(* Logix 5000 project; controller SX_V040001_C001 vendor 1 type 14 code 77 rev 16.23; software revision 16.04; part 27 of 35 *)
(* tags used below, declared in another part *)
   ALL_KINDS : INT[90];
   loading : INT[19];
   METERING : INT[44];
   NOTDOS : INT[6];
   PARAMETER : INT[501];
   T_DELTA_EM_METER : TIMER;
(* MainProgram, continued *)

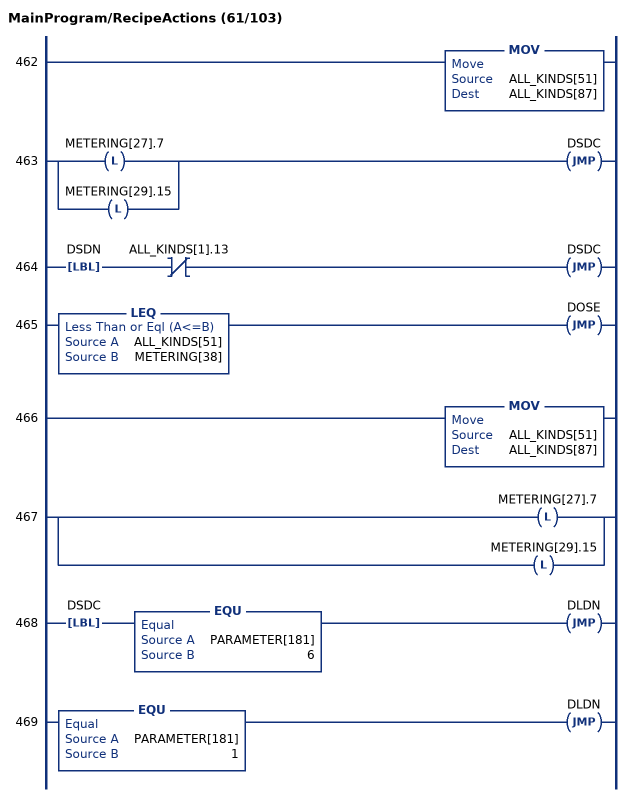
   [picture p595: MainProgram/RecipeActions rungs 462-469]
   462: MOV(ALL_KINDS[51],ALL_KINDS[87]);
   463: [OTL(METERING[27].7) ,OTL(METERING[29].15) ]JMP(DSDC);
   464: LBL(DSDN)XIO(ALL_KINDS[1].13)JMP(DSDC);
   465: LEQ(ALL_KINDS[51],METERING[38])JMP(DOSE);
   466: MOV(ALL_KINDS[51],ALL_KINDS[87]);
   467: [OTL(METERING[27].7) ,OTL(METERING[29].15) ];
   468: LBL(DSDC)EQU(PARAMETER[181],6)JMP(DLDN);
   469: EQU(PARAMETER[181],1)JMP(DLDN);
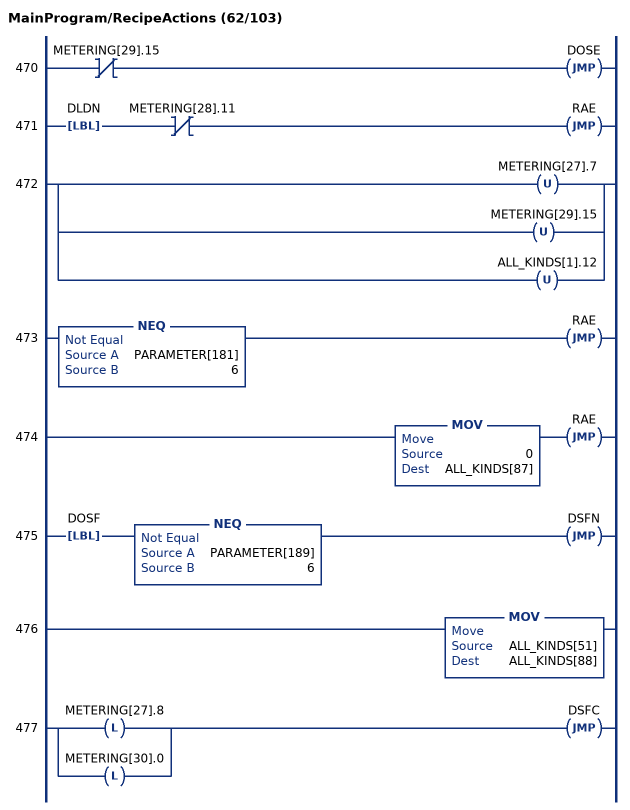
   470: XIO(METERING[29].15)JMP(DOSE);
   471: LBL(DLDN)XIO(METERING[28].11)JMP(RAE);
   472: [OTU(METERING[27].7) ,OTU(METERING[29].15) ,OTU(ALL_KINDS[1].12) ];
   473: NEQ(PARAMETER[181],6)JMP(RAE);
   474: MOV(0,ALL_KINDS[87])JMP(RAE);
   475: LBL(DOSF)NEQ(PARAMETER[189],6)JMP(DSFN);
   476: MOV(ALL_KINDS[51],ALL_KINDS[88]);
   477: [OTL(METERING[27].8) ,OTL(METERING[30].0) ]JMP(DSFC);
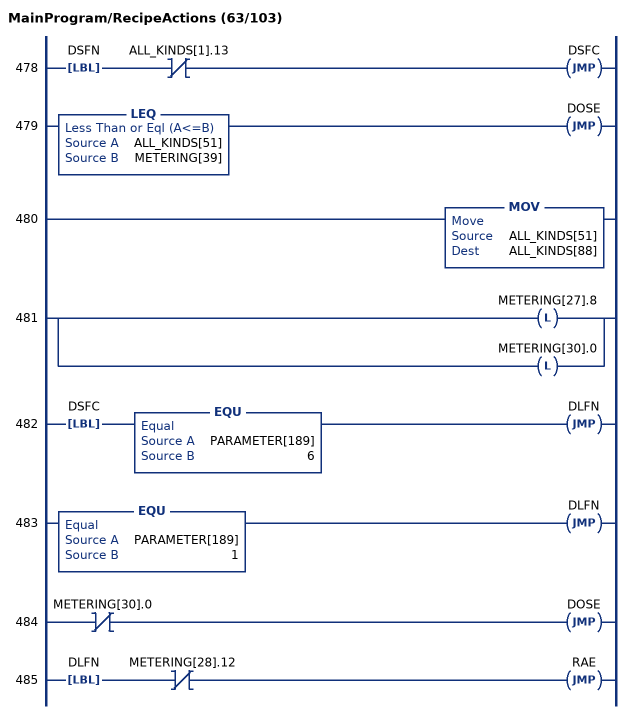
   478: LBL(DSFN)XIO(ALL_KINDS[1].13)JMP(DSFC);
   479: LEQ(ALL_KINDS[51],METERING[39])JMP(DOSE);
   480: MOV(ALL_KINDS[51],ALL_KINDS[88]);
   481: [OTL(METERING[27].8) ,OTL(METERING[30].0) ];
   482: LBL(DSFC)EQU(PARAMETER[189],6)JMP(DLFN);
   483: EQU(PARAMETER[189],1)JMP(DLFN);
   484: XIO(METERING[30].0)JMP(DOSE);
   485: LBL(DLFN)XIO(METERING[28].12)JMP(RAE);
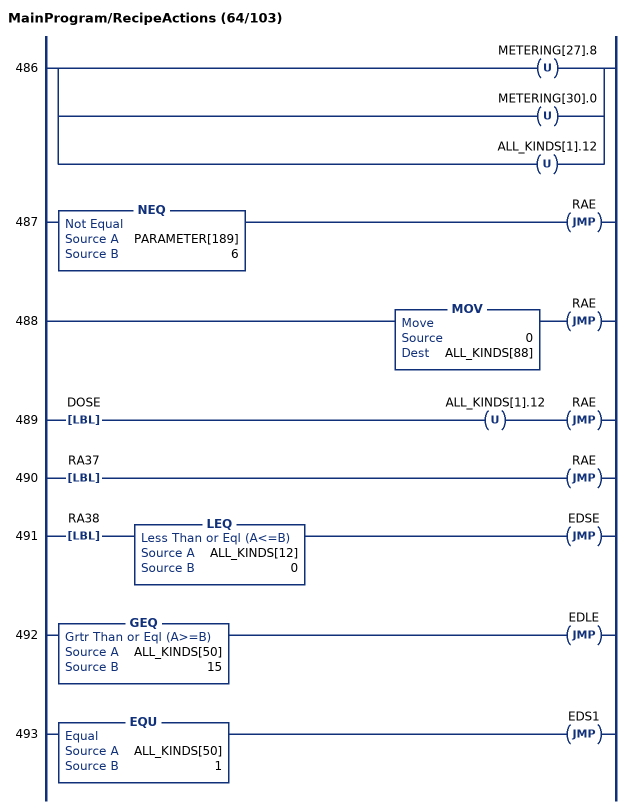
   486: [OTU(METERING[27].8) ,OTU(METERING[30].0) ,OTU(ALL_KINDS[1].12) ];
   487: NEQ(PARAMETER[189],6)JMP(RAE);
   488: MOV(0,ALL_KINDS[88])JMP(RAE);
   489: LBL(DOSE)OTU(ALL_KINDS[1].12)JMP(RAE);
   490: LBL(RA37)JMP(RAE);
   491: LBL(RA38)LEQ(ALL_KINDS[12],0)JMP(EDSE);
   492: GEQ(ALL_KINDS[50],15)JMP(EDLE);
   493: EQU(ALL_KINDS[50],1)JMP(EDS1);
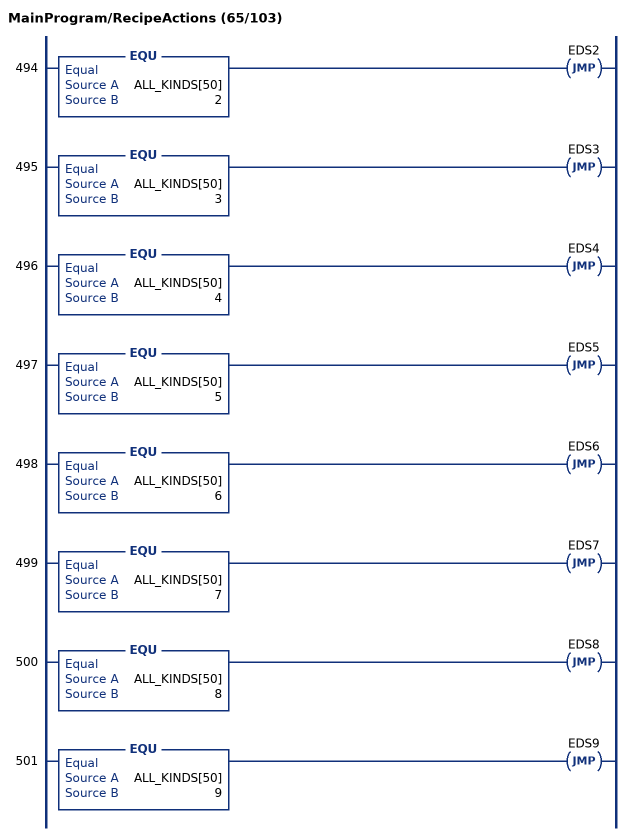
   494: EQU(ALL_KINDS[50],2)JMP(EDS2);
   495: EQU(ALL_KINDS[50],3)JMP(EDS3);
   496: EQU(ALL_KINDS[50],4)JMP(EDS4);
   497: EQU(ALL_KINDS[50],5)JMP(EDS5);
   498: EQU(ALL_KINDS[50],6)JMP(EDS6);
   499: EQU(ALL_KINDS[50],7)JMP(EDS7);
   500: EQU(ALL_KINDS[50],8)JMP(EDS8);
   501: EQU(ALL_KINDS[50],9)JMP(EDS9);
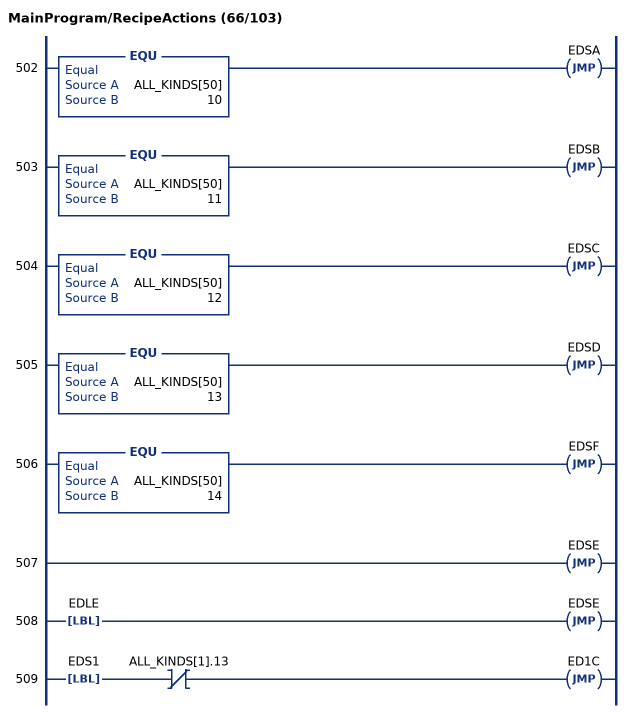
   502: EQU(ALL_KINDS[50],10)JMP(EDSA);
   503: EQU(ALL_KINDS[50],11)JMP(EDSB);
   504: EQU(ALL_KINDS[50],12)JMP(EDSC);
   505: EQU(ALL_KINDS[50],13)JMP(EDSD);
   506: EQU(ALL_KINDS[50],14)JMP(EDSF);
   507: JMP(EDSE);
   508: LBL(EDLE)JMP(EDSE);
   509: LBL(EDS1)XIO(ALL_KINDS[1].13)JMP(ED1C);
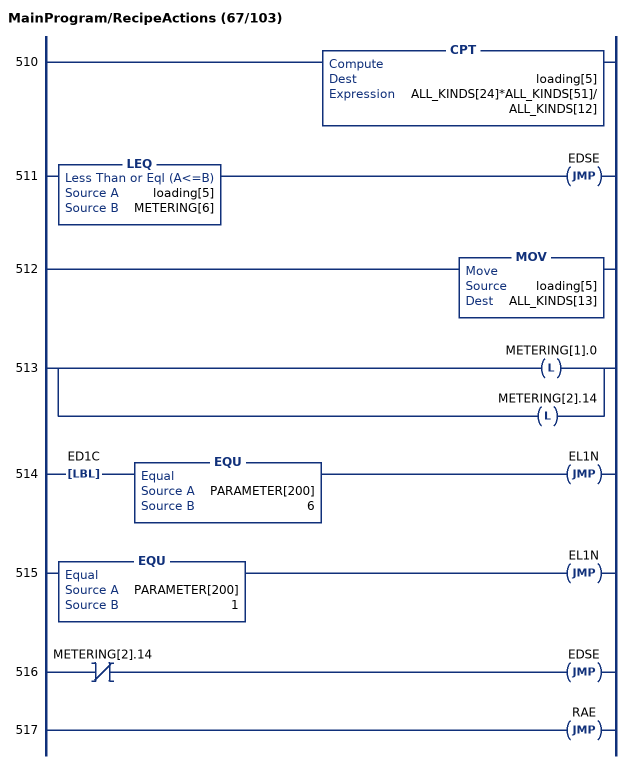
   510: CPT(loading[5],ALL_KINDS[24]*ALL_KINDS[51]/ALL_KINDS[12]);
   511: LEQ(loading[5],METERING[6])JMP(EDSE);
   512: MOV(loading[5],ALL_KINDS[13]);
   513: [OTL(METERING[1].0) ,OTL(METERING[2].14) ];
   514: LBL(ED1C)EQU(PARAMETER[200],6)JMP(EL1N);
   515: EQU(PARAMETER[200],1)JMP(EL1N);
   516: XIO(METERING[2].14)JMP(EDSE);
   517: JMP(RAE);
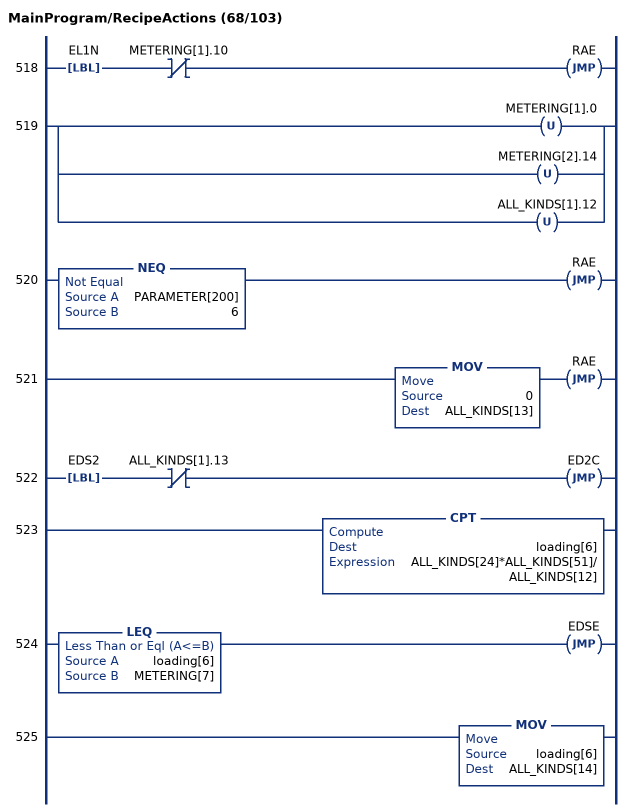
   518: LBL(EL1N)XIO(METERING[1].10)JMP(RAE);
   519: [OTU(METERING[1].0) ,OTU(METERING[2].14) ,OTU(ALL_KINDS[1].12) ];
   520: NEQ(PARAMETER[200],6)JMP(RAE);
   521: MOV(0,ALL_KINDS[13])JMP(RAE);
   522: LBL(EDS2)XIO(ALL_KINDS[1].13)JMP(ED2C);
   523: CPT(loading[6],ALL_KINDS[24]*ALL_KINDS[51]/ALL_KINDS[12]);
   524: LEQ(loading[6],METERING[7])JMP(EDSE);
   525: MOV(loading[6],ALL_KINDS[14]);
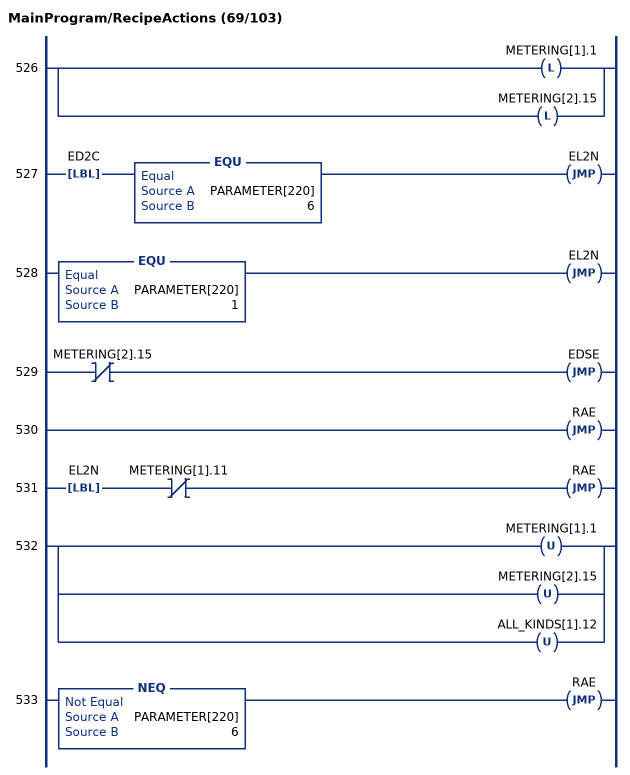
   526: [OTL(METERING[1].1) ,OTL(METERING[2].15) ];
   527: LBL(ED2C)EQU(PARAMETER[220],6)JMP(EL2N);
   528: EQU(PARAMETER[220],1)JMP(EL2N);
   529: XIO(METERING[2].15)JMP(EDSE);
   530: JMP(RAE);
   531: LBL(EL2N)XIO(METERING[1].11)JMP(RAE);
   532: [OTU(METERING[1].1) ,OTU(METERING[2].15) ,OTU(ALL_KINDS[1].12) ];
   533: NEQ(PARAMETER[220],6)JMP(RAE);
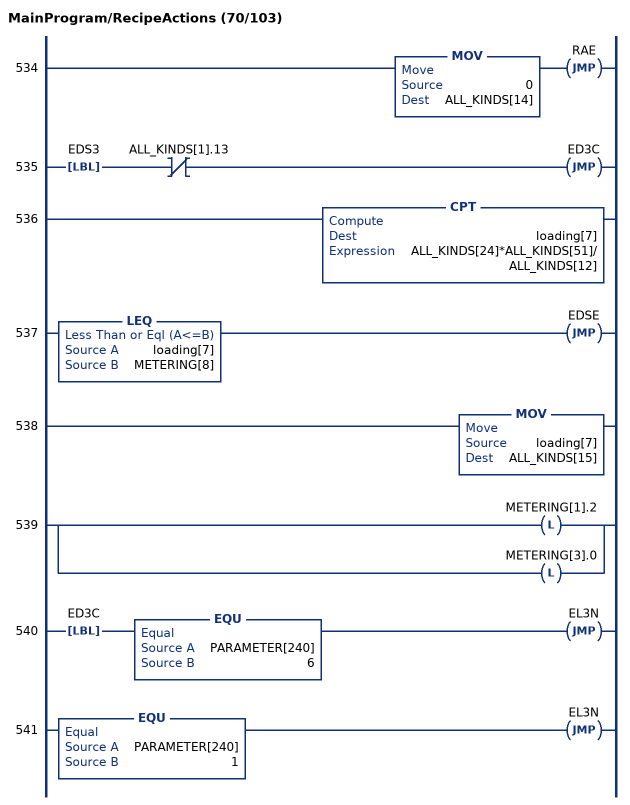
   534: MOV(0,ALL_KINDS[14])JMP(RAE);
   535: LBL(EDS3)XIO(ALL_KINDS[1].13)JMP(ED3C);
   536: CPT(loading[7],ALL_KINDS[24]*ALL_KINDS[51]/ALL_KINDS[12]);
   537: LEQ(loading[7],METERING[8])JMP(EDSE);
   538: MOV(loading[7],ALL_KINDS[15]);
   539: [OTL(METERING[1].2) ,OTL(METERING[3].0) ];
   540: LBL(ED3C)EQU(PARAMETER[240],6)JMP(EL3N);
   541: EQU(PARAMETER[240],1)JMP(EL3N);
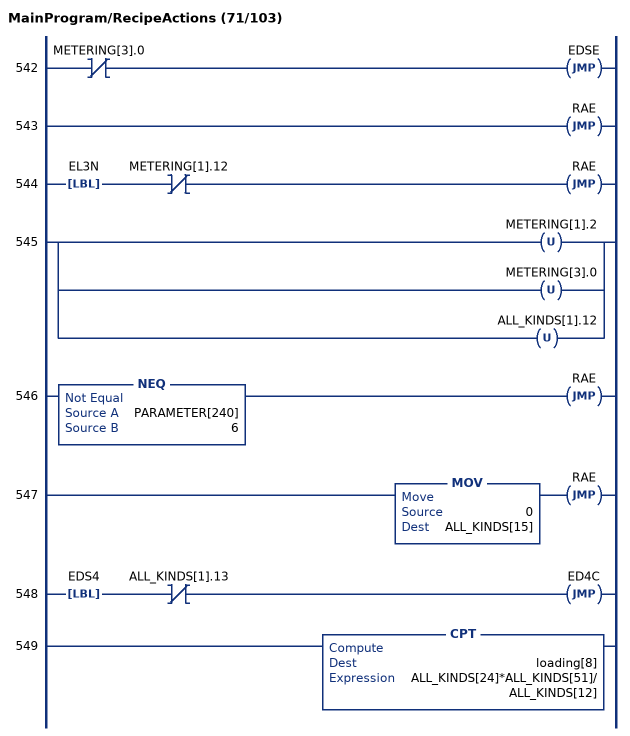
   542: XIO(METERING[3].0)JMP(EDSE);
   543: JMP(RAE);
   544: LBL(EL3N)XIO(METERING[1].12)JMP(RAE);
   545: [OTU(METERING[1].2) ,OTU(METERING[3].0) ,OTU(ALL_KINDS[1].12) ];
   546: NEQ(PARAMETER[240],6)JMP(RAE);
   547: MOV(0,ALL_KINDS[15])JMP(RAE);
   548: LBL(EDS4)XIO(ALL_KINDS[1].13)JMP(ED4C);
   549: CPT(loading[8],ALL_KINDS[24]*ALL_KINDS[51]/ALL_KINDS[12]);
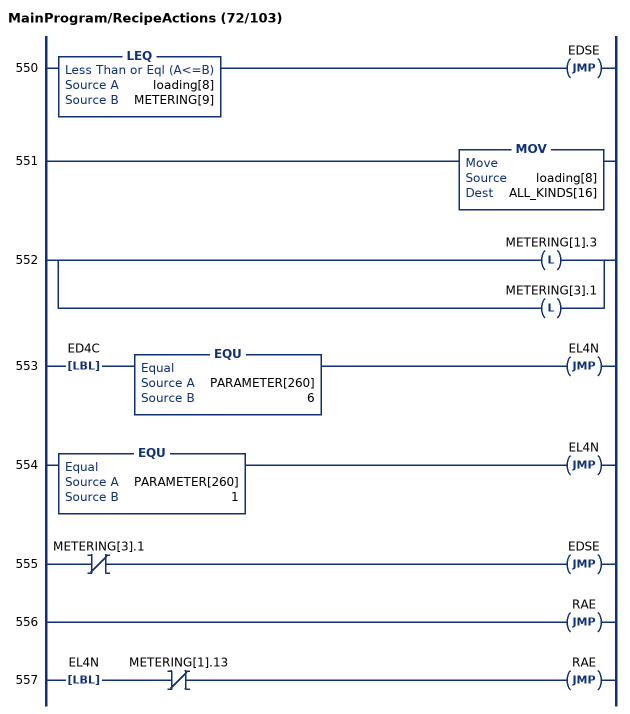
   550: LEQ(loading[8],METERING[9])JMP(EDSE);
   551: MOV(loading[8],ALL_KINDS[16]);
   552: [OTL(METERING[1].3) ,OTL(METERING[3].1) ];
   553: LBL(ED4C)EQU(PARAMETER[260],6)JMP(EL4N);
   554: EQU(PARAMETER[260],1)JMP(EL4N);
   555: XIO(METERING[3].1)JMP(EDSE);
   556: JMP(RAE);
   557: LBL(EL4N)XIO(METERING[1].13)JMP(RAE);
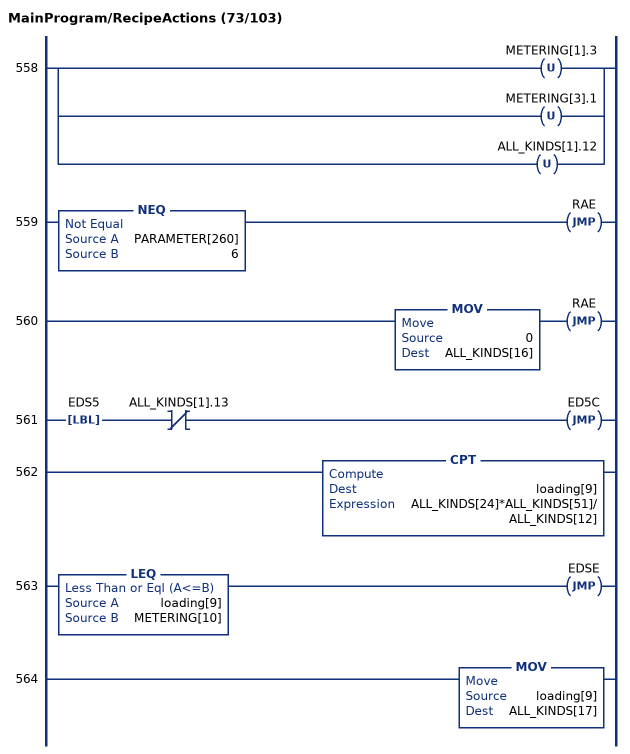
   558: [OTU(METERING[1].3) ,OTU(METERING[3].1) ,OTU(ALL_KINDS[1].12) ];
   559: NEQ(PARAMETER[260],6)JMP(RAE);
   560: MOV(0,ALL_KINDS[16])JMP(RAE);
   561: LBL(EDS5)XIO(ALL_KINDS[1].13)JMP(ED5C);
   562: CPT(loading[9],ALL_KINDS[24]*ALL_KINDS[51]/ALL_KINDS[12]);
   563: LEQ(loading[9],METERING[10])JMP(EDSE);
   564: MOV(loading[9],ALL_KINDS[17]);
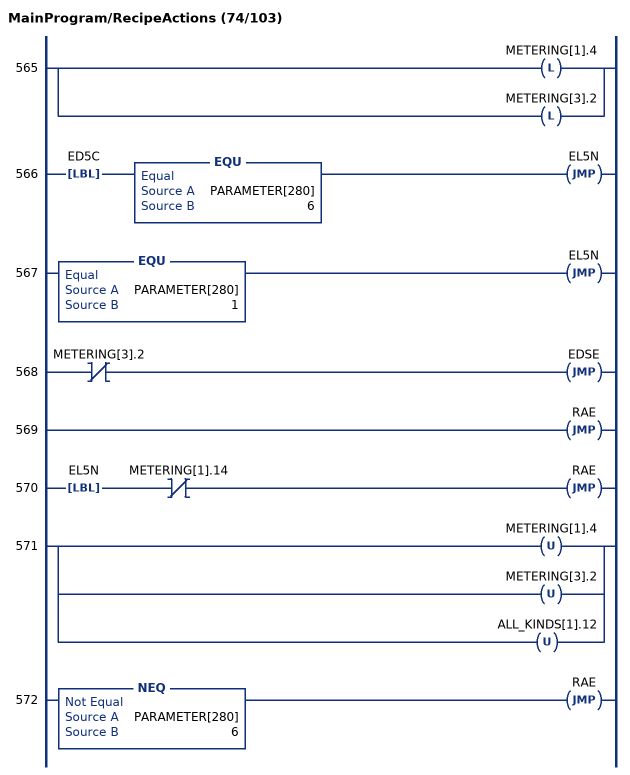
   565: [OTL(METERING[1].4) ,OTL(METERING[3].2) ];
   566: LBL(ED5C)EQU(PARAMETER[280],6)JMP(EL5N);
   567: EQU(PARAMETER[280],1)JMP(EL5N);
   568: XIO(METERING[3].2)JMP(EDSE);
   569: JMP(RAE);
   570: LBL(EL5N)XIO(METERING[1].14)JMP(RAE);
   571: [OTU(METERING[1].4) ,OTU(METERING[3].2) ,OTU(ALL_KINDS[1].12) ];
   572: NEQ(PARAMETER[280],6)JMP(RAE);
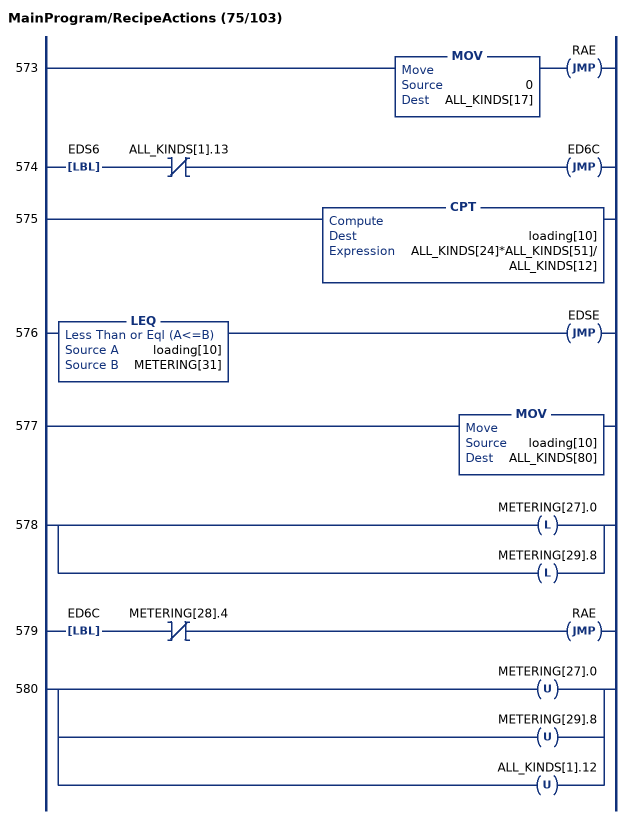
   573: MOV(0,ALL_KINDS[17])JMP(RAE);
   574: LBL(EDS6)XIO(ALL_KINDS[1].13)JMP(ED6C);
   575: CPT(loading[10],ALL_KINDS[24]*ALL_KINDS[51]/ALL_KINDS[12]);
   576: LEQ(loading[10],METERING[31])JMP(EDSE);
   577: MOV(loading[10],ALL_KINDS[80]);
   578: [OTL(METERING[27].0) ,OTL(METERING[29].8) ];
   579: LBL(ED6C)XIO(METERING[28].4)JMP(RAE);
   580: [OTU(METERING[27].0) ,OTU(METERING[29].8) ,OTU(ALL_KINDS[1].12) ];
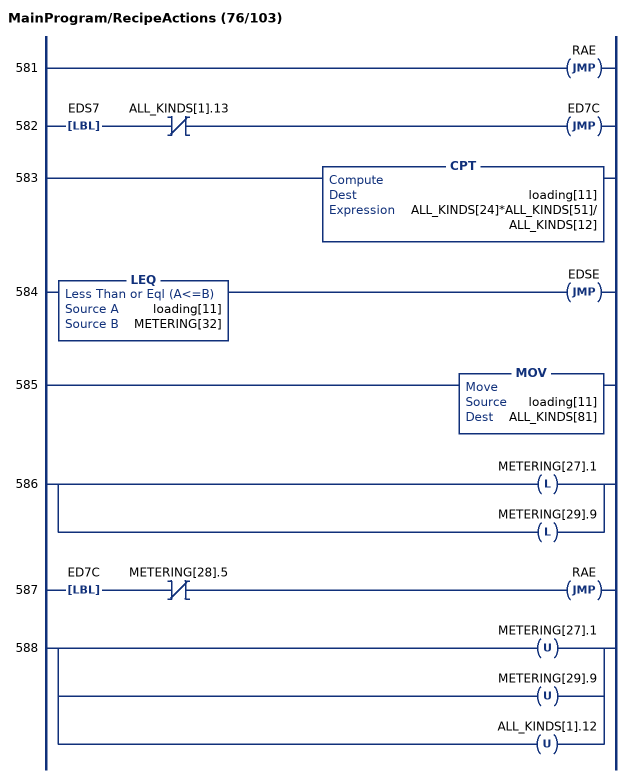
   581: JMP(RAE);
   582: LBL(EDS7)XIO(ALL_KINDS[1].13)JMP(ED7C);
   583: CPT(loading[11],ALL_KINDS[24]*ALL_KINDS[51]/ALL_KINDS[12]);
   584: LEQ(loading[11],METERING[32])JMP(EDSE);
   585: MOV(loading[11],ALL_KINDS[81]);
   586: [OTL(METERING[27].1) ,OTL(METERING[29].9) ];
   587: LBL(ED7C)XIO(METERING[28].5)JMP(RAE);
   588: [OTU(METERING[27].1) ,OTU(METERING[29].9) ,OTU(ALL_KINDS[1].12) ];
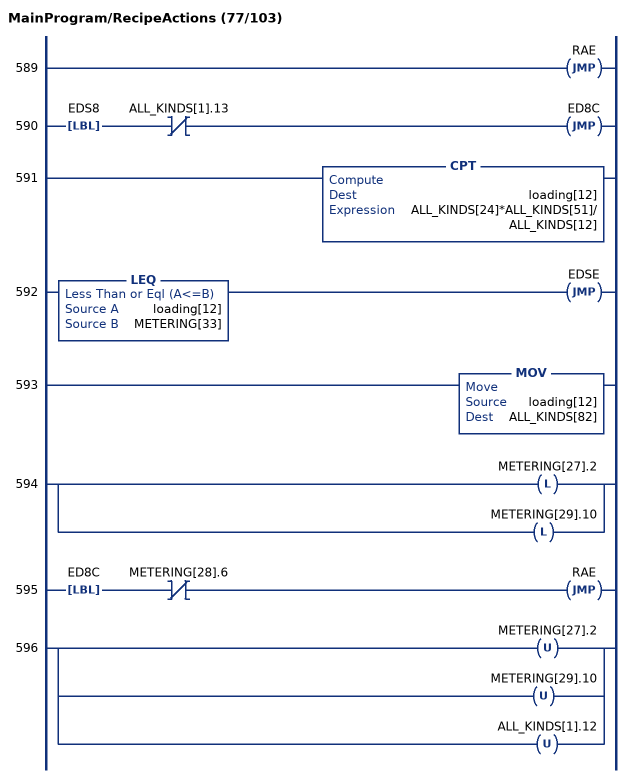
   589: JMP(RAE);
   590: LBL(EDS8)XIO(ALL_KINDS[1].13)JMP(ED8C);
   591: CPT(loading[12],ALL_KINDS[24]*ALL_KINDS[51]/ALL_KINDS[12]);
   592: LEQ(loading[12],METERING[33])JMP(EDSE);
   593: MOV(loading[12],ALL_KINDS[82]);
   594: [OTL(METERING[27].2) ,OTL(METERING[29].10) ];
   595: LBL(ED8C)XIO(METERING[28].6)JMP(RAE);
   596: [OTU(METERING[27].2) ,OTU(METERING[29].10) ,OTU(ALL_KINDS[1].12) ];
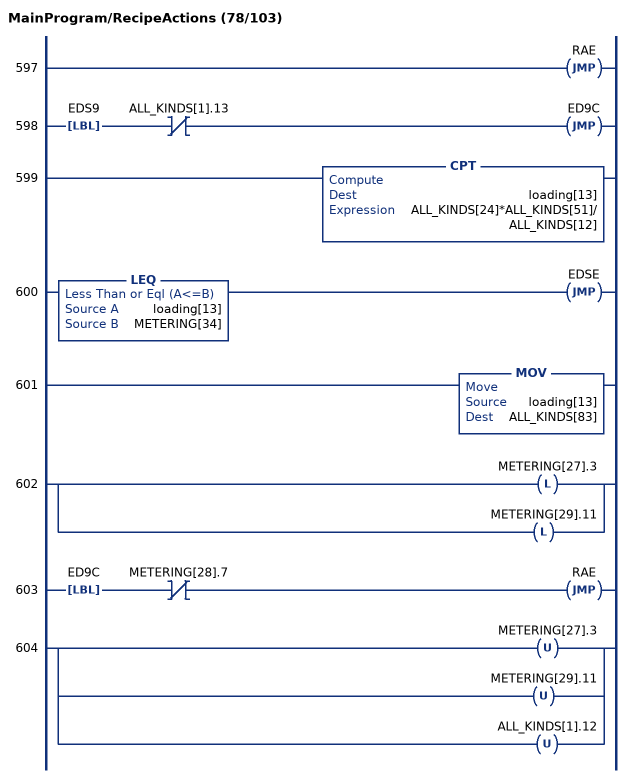
   597: JMP(RAE);
   598: LBL(EDS9)XIO(ALL_KINDS[1].13)JMP(ED9C);
   599: CPT(loading[13],ALL_KINDS[24]*ALL_KINDS[51]/ALL_KINDS[12]);
   600: LEQ(loading[13],METERING[34])JMP(EDSE);
   601: MOV(loading[13],ALL_KINDS[83]);
   602: [OTL(METERING[27].3) ,OTL(METERING[29].11) ];
   603: LBL(ED9C)XIO(METERING[28].7)JMP(RAE);
   604: [OTU(METERING[27].3) ,OTU(METERING[29].11) ,OTU(ALL_KINDS[1].12) ];
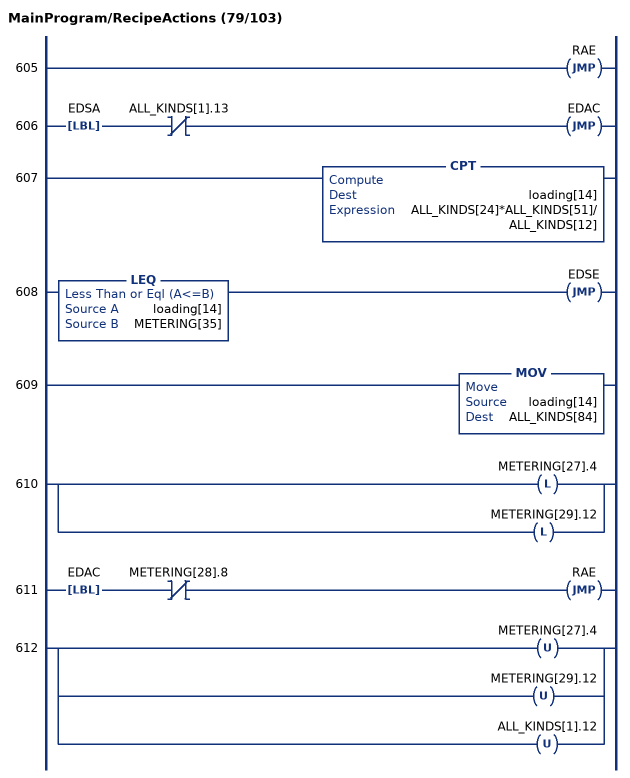
   605: JMP(RAE);
   606: LBL(EDSA)XIO(ALL_KINDS[1].13)JMP(EDAC);
   607: CPT(loading[14],ALL_KINDS[24]*ALL_KINDS[51]/ALL_KINDS[12]);
   608: LEQ(loading[14],METERING[35])JMP(EDSE);
   609: MOV(loading[14],ALL_KINDS[84]);
   610: [OTL(METERING[27].4) ,OTL(METERING[29].12) ];
   611: LBL(EDAC)XIO(METERING[28].8)JMP(RAE);
   612: [OTU(METERING[27].4) ,OTU(METERING[29].12) ,OTU(ALL_KINDS[1].12) ];
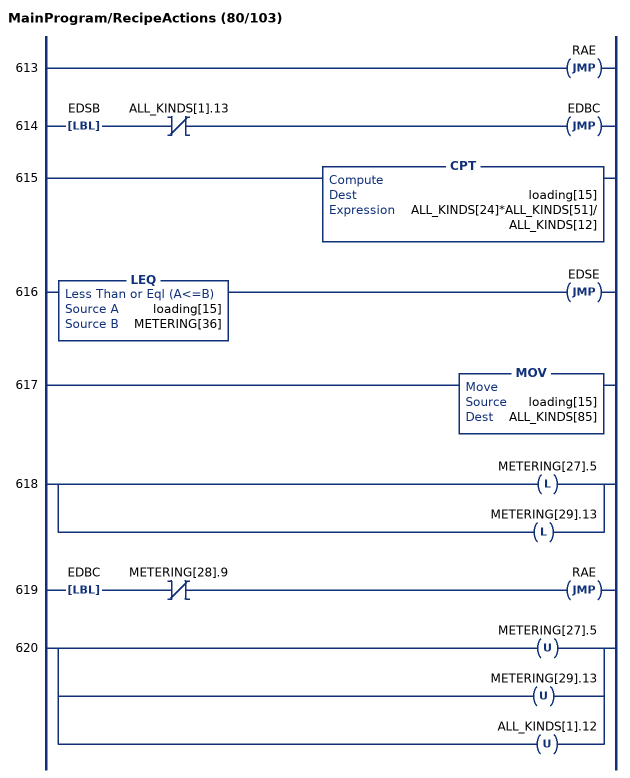
   613: JMP(RAE);
   614: LBL(EDSB)XIO(ALL_KINDS[1].13)JMP(EDBC);
   615: CPT(loading[15],ALL_KINDS[24]*ALL_KINDS[51]/ALL_KINDS[12]);
   616: LEQ(loading[15],METERING[36])JMP(EDSE);
   617: MOV(loading[15],ALL_KINDS[85]);
   618: [OTL(METERING[27].5) ,OTL(METERING[29].13) ];
   619: LBL(EDBC)XIO(METERING[28].9)JMP(RAE);
   620: [OTU(METERING[27].5) ,OTU(METERING[29].13) ,OTU(ALL_KINDS[1].12) ];
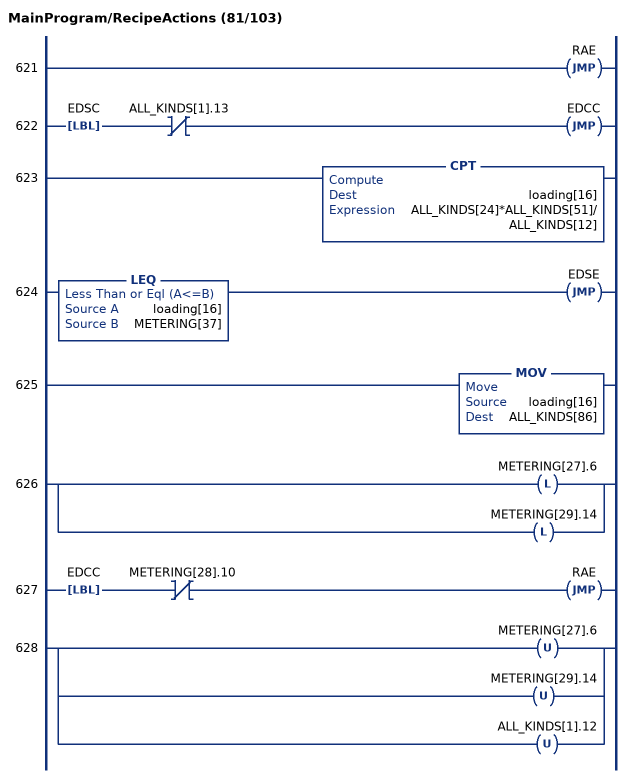
   621: JMP(RAE);
   622: LBL(EDSC)XIO(ALL_KINDS[1].13)JMP(EDCC);
   623: CPT(loading[16],ALL_KINDS[24]*ALL_KINDS[51]/ALL_KINDS[12]);
   624: LEQ(loading[16],METERING[37])JMP(EDSE);
   625: MOV(loading[16],ALL_KINDS[86]);
   626: [OTL(METERING[27].6) ,OTL(METERING[29].14) ];
   627: LBL(EDCC)XIO(METERING[28].10)JMP(RAE);
   628: [OTU(METERING[27].6) ,OTU(METERING[29].14) ,OTU(ALL_KINDS[1].12) ];
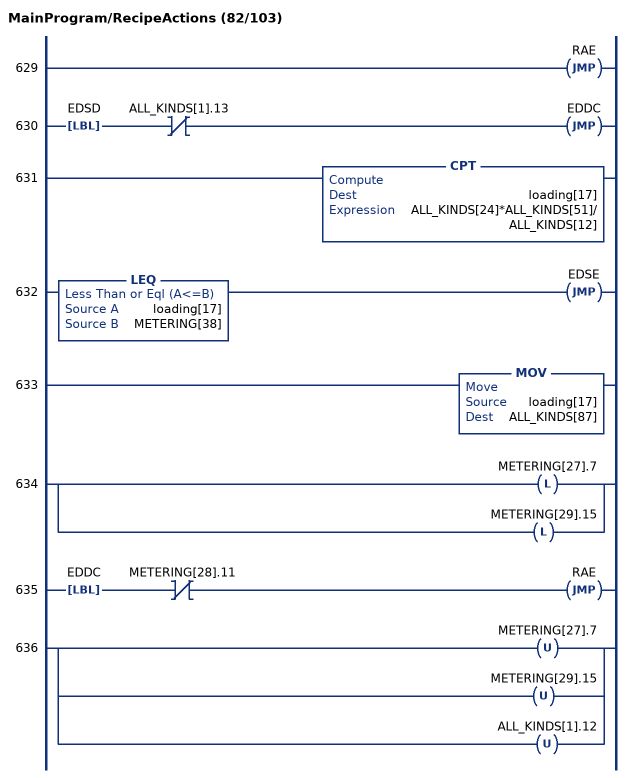
   629: JMP(RAE);
   630: LBL(EDSD)XIO(ALL_KINDS[1].13)JMP(EDDC);
   631: CPT(loading[17],ALL_KINDS[24]*ALL_KINDS[51]/ALL_KINDS[12]);
   632: LEQ(loading[17],METERING[38])JMP(EDSE);
   633: MOV(loading[17],ALL_KINDS[87]);
   634: [OTL(METERING[27].7) ,OTL(METERING[29].15) ];
   635: LBL(EDDC)XIO(METERING[28].11)JMP(RAE);
   636: [OTU(METERING[27].7) ,OTU(METERING[29].15) ,OTU(ALL_KINDS[1].12) ];
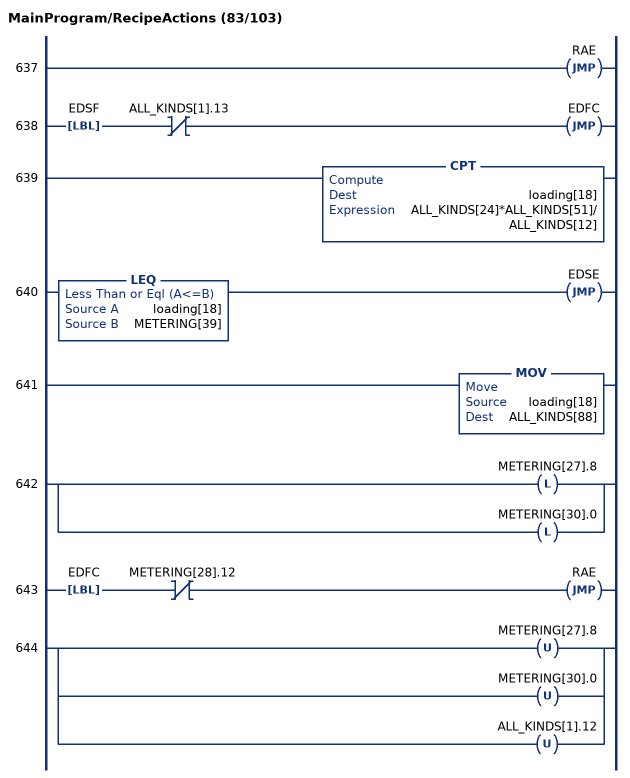
   637: JMP(RAE);
   638: LBL(EDSF)XIO(ALL_KINDS[1].13)JMP(EDFC);
   639: CPT(loading[18],ALL_KINDS[24]*ALL_KINDS[51]/ALL_KINDS[12]);
   640: LEQ(loading[18],METERING[39])JMP(EDSE);
   641: MOV(loading[18],ALL_KINDS[88]);
   642: [OTL(METERING[27].8) ,OTL(METERING[30].0) ];
   643: LBL(EDFC)XIO(METERING[28].12)JMP(RAE);
   644: [OTU(METERING[27].8) ,OTU(METERING[30].0) ,OTU(ALL_KINDS[1].12) ];
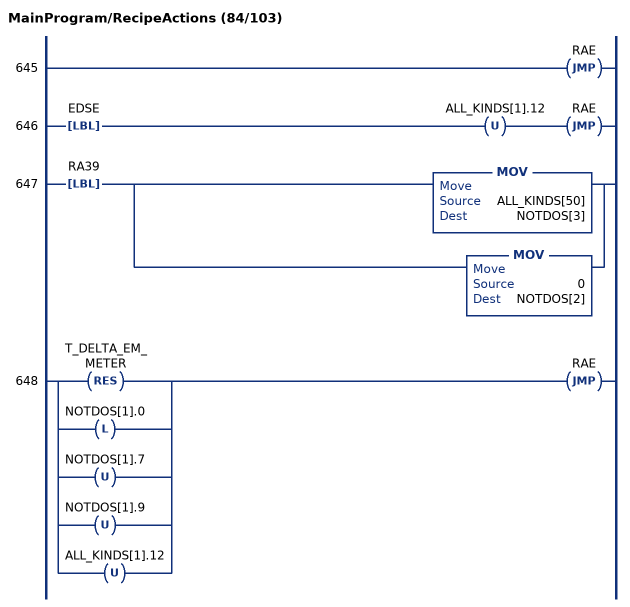
   645: JMP(RAE);
   646: LBL(EDSE)OTU(ALL_KINDS[1].12)JMP(RAE);
   647: LBL(RA39)[MOV(ALL_KINDS[50],NOTDOS[3]) ,MOV(0,NOTDOS[2]) ];
   648: [RES(T_DELTA_EM_METER) ,OTL(NOTDOS[1].0) ,OTU(NOTDOS[1].7) ,OTU(NOTDOS[1].9) ,OTU(ALL_KINDS[1].12) ]JMP(RAE);
